(* PLC project SharedBoxFixture, greenforge-labs codescribe-fixture 1 *)
(* stored: creationDateTime 2020-01-01T00:00:00 *)

PROGRAM FBD_SHARED
  VAR
    fbTimer : TON;
  END_VAR

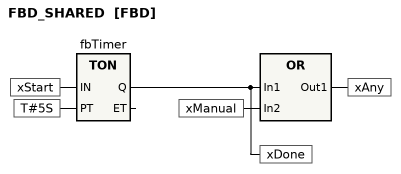
(* FBD diagram, written out as Structured Text *)
fbTimer(IN := xStart, PT := T#5S);
xDone := fbTimer.Q;
xAny := fbTimer.Q OR xManual;
END_PROGRAM
